PROGRAM MAIN
VAR
	{attribute wpf [Container(Layout.Tabs)]}
	App :stPrograms;
END_VAR

App.EmailSender();
App.Sorting();
App.Data();
App.TextMsg();
App.RestCall();

END_PROGRAM

(* stored: Version 1.1.0.1, ProductVersion 3.1.4024.5
   POU MAIN: Id {2aec7386-fec2-4299-8c2e-88bb20ee3274}, SpecialFunc None *)
